INTERFACE ITF_DBAdaptor

METHOD SQL_Delete : DB_FunctionResult
VAR_INPUT
	SQL : STRING(255);
END_VAR
END_METHOD

PROPERTY TimeOut : TIME
GET
END_GET
SET
END_SET
END_PROPERTY

PROPERTY sNetID : string(23)
SET
END_SET
GET
END_GET
END_PROPERTY

METHOD SQL_Insert : DB_FunctionResult
VAR_INPUT
	SQL 				: STRING(255);
END_VAR
END_METHOD

METHOD SQL_Select : DB_FunctionResult
VAR_INPUT
	SQL 				: STRING(255);
	START_INDEX			: UDINT;
	ROWS				: UDINT;
	ROW_DATA_BYTES		: UDINT;
	ptr_ReceiveBuffer	: POINTER TO BYTE;
END_VAR
END_METHOD

PROPERTY udiDatabase_ID : UDINT
SET
END_SET
GET
END_GET
END_PROPERTY

END_INTERFACE

(* stored: Version 1.1.0.1, ProductVersion 3.1.0.36
   Itf ITF_DBAdaptor: Id {9f1b48f4-eeab-41cf-aa48-0de36856ceaf}
   Method SQL_Delete: Id {0fbb7eef-5b1d-4ce3-9a20-27f9497c2b6f}
   Property TimeOut: Id {5779eafa-16cf-470a-8f85-7ccb89d20314}
   Get Get: Id {3c7c7727-a7d6-4cbb-8131-c3f33dedc97d}
   Set Set: Id {81c24d5a-eb28-4a7d-9faa-7afa6d22e4c4}
   Property sNetID: Id {6218a16c-d9f3-41b9-bb01-140403b9e4c6}
   Set Set: Id {821fd5a2-7ab2-4f39-8241-5e34a7276c51}
   Get Get: Id {f3d3ea48-2b82-4d77-8095-103ff0a43b18}
   Method SQL_Insert: Id {78ccc74b-ce47-4f46-be9e-3db2490b5857}
   Method SQL_Select: Id {e40e14ef-015a-4862-afd8-c63b79cb4a71}
   Property udiDatabase_ID: Id {e894097f-8ff3-442b-98a0-e40afe89fbbc}
   Set Set: Id {2b84286a-d965-4af1-a8e4-0fbc497a20e3}
   Get Get: Id {716134e7-56b7-43fc-8b20-ce1f2c2effb9} *)
